# EPICS StreamDevice protocol: protocols/ao420fmc.proto
Terminator = LF;
ExtraInput = Ignore;

setRange {
	out "dac_range_0\$1 %d";
	in;
}
